(* PLC project édi, Bombardier Transportation 1131-TOOL 3.0.0.2 *)
(* stored: companyURL www.kw-software.com, creationDateTime 2015-03-05T11:10:42, version 1425550242, modificationDateTime 2015-03-05T11:10:42 *)

PROGRAM th_X_Trip
  VAR_INPUT
    f_X : INT;
    f_Module_Error : BOOL;
    f_Channel_Error : BOOL;
    tx_X_Logic_Trip : BOOL;
  END_VAR
  VAR
    K_X_Min : INT := -55;
  END_VAR
  VAR_OUTPUT
    tx_X_trip : BOOL;
  END_VAR
  VAR
    k_X_Max : INT := 125;
  END_VAR

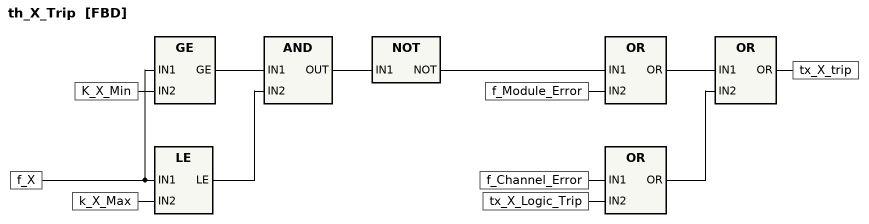
(* FBD diagram, written out as Structured Text *)
tx_X_trip := NOT (f_X >= K_X_Min AND f_X <= k_X_Max) OR f_Module_Error OR f_Channel_Error OR tx_X_Logic_Trip;
END_PROGRAM
